PROGRAM MAIN_1
VAR
END_VAR

P_Box_Controll();

END_PROGRAM

(* stored: Version 1.1.0.1, ProductVersion 3.1.4024.12
   POU MAIN_1: Id {08577184-405e-4799-aa4b-48577b931b68}, SpecialFunc None *)
